(* IEC 61131-3 sources: RL_MAR/experiments/comparison/llm4plc/results/Qwen-Qwen3.5-9B_20260506_150728/20260506_163730, 1 file *)

(* ---- generated_code_iteration_0.st ---- *)
START_ST
FUNCTION_BLOCK FlowerArrangingMachine
VAR_INPUT
    FlowerTypeSensor : INT; (* Input for detecting flower type *)
    FlowerColorSensor : INT; (* Input for detecting flower color *)
END_VAR
VAR_OUTPUT
    ArrangingMechanism : INT; (* Output for controlling arranging mechanism *)
    ConveyorBelt : BOOL; (* Output for controlling conveyor belt *)
END_VAR
VAR
    (* No internal variables strictly required as logic is direct mapping *)
END_VAR

(* STATE 0: EVALUATE_AND_UPDATE *)
(* Action: Read FlowerTypeSensor and FlowerColorSensor *)
(* Action: Calculate the required ArrangingMechanism value based on the combination *)
(* Action: Update ArrangingMechanism output *)
(* Action: Calculate ConveyorBelt status based on the new ArrangingMechanism value *)
(* Action: Update ConveyorBelt output *)

(* Logic to set ArrangingMechanism based on FlowerTypeSensor and FlowerColorSensor *)
IF FlowerTypeSensor = 1 AND FlowerColorSensor = 1 THEN
    ArrangingMechanism := 1; (* Red type 1 flower *)
ELSIF FlowerTypeSensor = 1 AND FlowerColorSensor = 2 THEN
    ArrangingMechanism := 2; (* Blue type 1 flower *)
ELSIF FlowerTypeSensor = 2 AND FlowerColorSensor = 1 THEN
    ArrangingMechanism := 3; (* Red type 2 flower *)
ELSIF FlowerTypeSensor = 2 AND FlowerColorSensor = 2 THEN
    ArrangingMechanism := 4; (* Blue type 2 flower *)
ELSE
    ArrangingMechanism := 0; (* Any other combination *)
END_IF;

(* Logic to set ConveyorBelt based on ArrangingMechanism *)
IF ArrangingMechanism <> 0 THEN
    ConveyorBelt := TRUE;
ELSE
    ConveyorBelt := FALSE;
END_IF;

END_FUNCTION_BLOCK
END_ST
